// use slot attribute larger than 49990, which is the default one, if it depends on variable in other file
{attribute 'global_init_slot' := '49991'} 
{attribute 'qualified_only'}
VAR_GLOBAL CONSTANT 

(* 
% setup arm
% 1        0      0   q1      0
% 2        90     a2   0      q2
% 3        -90     0   0       d4+q3
% 4        0       0   q4      0
% 5        -90      0   q5      0
*)
g_setupA2:ARRAY[1..4] OF LREAL:=[0.019,0.136, 0.136, 0.1825 ];
g_setupD4:ARRAY[1..4] OF LREAL:=[0.5205,0.3545, 0.3545, 0.5205 ];

//alpha,a,d,theta	
g_setupArmDH:ARRAY[1..5,1..4] OF LREAL  :=[   0,   0,   0,     0,
											PI/2,  g_setupA2[1],   0,      0,
											-PI/2,  0,   0,       g_setupD4[2],
											0,       0,   0,      0,
											-PI/2,   0,   0,      0];
									   
END_VAR

(* stored: Version 1.1.0.1, ProductVersion 3.1.4024.12
   GVL GVL_SetupArmKinematic: Id {51b5e92c-cdd9-424e-87d2-379444a190f7} *)
